// Mitsubishi GX Works2 project: FunctionBLK_ctu_ctd   PLC: Q03UDV

// task Task_01 (event TRUE, interval 0, priority 31): POU_01

PROGRAM POU_01
VAR
  CTD_1 : CTD;
  counter1 : BOOL;
  CTU_1 : CTU;
  counter2 : BOOL;
  CTU_2 : CTU;
  TP_1 : TP;
  TIMER1 : BOOL;
  TON_1 : TON;
  TIMER2 : BOOL;
  TOF_1 : TOF;
  TOF_2 : TOF;
  TIMER3 : BOOL;
  TimerTP : TIME;
  TimeON : TIME;
  TimeOFF : TIME;
END_VAR
(* structured ladder/FBD written out as ST: instructions are called as NAME(EN, inputs, outputs); _pN, _eN, _tN stand for wires *)
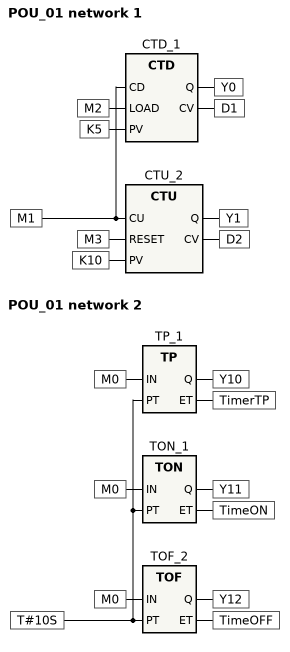
(* network 1 *)
CTD_1(CD := M1, LOAD := M2, PV := K5, Q => Y0, CV => D1);
CTU_2(CU := M1, RESET := M3, PV := K10, Q => Y1, CV => D2);
(* network 2 *)
TP_1(IN := M0, PT := T#10S, Q => Y10, ET => TimerTP);
TON_1(IN := M0, PT := T#10S, Q => Y11, ET => TimeON);
TOF_2(IN := M0, PT := T#10S, Q => Y12, ET => TimeOFF);
END_PROGRAM
